Fanuc KAREL source: ka00105.KL

PROGRAM KA00105
%STACKSIZE=65535
%PRIORITY=65535
%NOLOCKGROUP
-- UNRESOLVED DECLARATIONS (source type spelling not recovered)
-- SRC : TYPE_0x0013 (type_u16=0x0013)
-- DST : TYPE_0x0013 (type_u16=0x0013)
BEGIN
-- UNSAFE_SOURCE_IR line 7: field_offset(SRC,0) = 1065353216
-- UNRESOLVED_PC line 8 opcodes [49 4A] marker_code=20
END KA00105
